FUNCTION_BLOCK FB_Sample EXTENDS FB_Generic
VAR_INPUT
END_VAR
VAR_OUTPUT
END_VAR
VAR
	lamp			: BOOL;	
	eStates			: E_SampleStates := E_SampleStates.IDLE;;
	eStateTemp		: E_SampleStates := E_SampleStates.IDLE;
	iStateTemp		: INT;	
END_VAR

SUPER^();
IF NOT subscribed THEN
	GVL.PubSubService.Subscribe(E_Topics.SAMPLE_SUBSCRRIBE_1,THIS^);
	GVL.PubSubService.Subscribe(E_Topics.SAMPLE_SUBSCRRIBE_2,THIS^);
	GVL.PubSubService.Subscribe(E_Topics.SAMPLE_SUBSCRRIBE_3,THIS^);
END_IF
subscribed	:= TRUE;


sComponent_name		:= 'fb_sample';
iComponetID			:= 99;
strState	:= ParseStateToString();

(*
Description: 
the callback that will be invoked when there is a publish for what the subscriber was subscribed to.
*)
METHOD Callback
VAR_INPUT
	data : PubSubData;
END_VAR
CASE data.Topic OF
	E_Topics.SAMPLE_SUBSCRRIBE_1:
		ADSLOGSTR(msgCtrlMask:= ADSLOG_MSGTYPE_LOG,msgFmtStr:='get data from publish 1',strArg:='');
	E_Topics.SAMPLE_SUBSCRRIBE_2:
		ADSLOGSTR(msgCtrlMask:= ADSLOG_MSGTYPE_LOG,msgFmtStr:='get data from publish 2',strArg:='');
	E_Topics.SAMPLE_SUBSCRRIBE_3:
		ADSLOGSTR(msgCtrlMask:= ADSLOG_MSGTYPE_LOG,msgFmtStr:='get data from publish 3',strArg:='');		
END_CASE
END_METHOD

{attribute 'object_name' := 'M_Aborting'}
METHOD M_Aborting
CASE fbUnitModeManager.eModeStatus OF	
	ePMLProtUnitMode_Production, ePMLProtUnitMode_Manual:		
		lamp	:= FALSE;		
		M_StateComplete();
			
	ePMLProtUnitMode_Maintenance, ePMLUnitMode_Service:
		
		M_StateComplete();
END_CASE
END_METHOD

METHOD M_agingTest : BOOL
VAR_INPUT
	
END_VAR
END_METHOD

{attribute 'object_name' := 'M_Completing'}
METHOD M_Completing
CASE fbUnitModeManager.eModeStatus OF
	ePMLProtUnitMode_Production:
		;
END_CASE
END_METHOD

{attribute 'object_name' := 'M_Execute'}
METHOD M_Execute

CASE fbUnitModeManager.eModeStatus OF
	ePMLProtUnitMode_Production:		//Mode Production
		//////////////////////////////////////////////////////////timeout//////////////////////////////////////////	
		iStateTemp	:= eStateTemp;
		ton_timeout();
		IF eStateTemp=eStates THEN
			ton_timeout.IN	:=TRUE;
		ELSE
			ton_timeout.IN	:=FALSE;
			eStateTemp	:= eStates;	
//			ParseStateToString();
//			GenerateErrorMsg(errorType:='M',strState:=ParseStateToString(),moduleID:=100,iState	:= iStateTemp);
			IF ton_timeout.Q THEN
				RETURN;
			END_IF
		END_IF
		IF ton_timeout.Q THEN	
			ton_timeout.IN	:=FALSE;
			CASE eStates OF	
				E_SampleStates.ERROR:	
					alarm_temp.Message	:= GenerateErrorMsg(errorType:='M',strState:=strState,iState := iStateTemp,errorMsg:='in error state.');
				ELSE
				alarm_temp.Message	:= GenerateErrorMsg(errorType:='M',strState:=strState,iState := iStateTemp,errorMsg:='time out');
			END_CASE
			
//			CASE eStates OF		
//				E_SampleStates.IDLE:						
//					;
//				E_SampleStates.INIT:
//					;
//				E_SampleStates.WAIT_ON:
//					;
//				E_SampleStates.WAIT_OFF:
//					;			
//				E_SampleStates.ERROR:	
//					alarm_temp.Message	:= 'Sample in error state';
//				ELSE
//					alarm_temp.Message	:= 'UNKNOWN STATES in Sample module';
//			END_CASE
			IF eStates<>E_SampleStates.IDLE AND eStates<>E_SampleStates.WAIT_ON AND eStates<>E_SampleStates.WAIT_OFF THEN
				GVL.pml_adminAlarm.M_SetAlarm(stAdmin:=GVL.PackTags.Admin,stAlarm:=alarm_temp);
			END_IF
		END_IF
		
		CASE eStates OF 
				E_SampleStates.IDLE:
					ton_timeout.PT	:= T#1MS;						
					eStates	:= E_SampleStates.INIT;				
				E_SampleStates.INIT:
					ton_timeout.PT	:= T#1S;
					eStates	:= E_SampleStates.WAIT_ON; 
				E_SampleStates.DETECTION:
					ton_timeout.PT	:= T#3S;
				E_SampleStates.WAIT:
					ton_timeout.PT	:= T#200MS;					
				E_SampleStates.WAIT_ON:
					lamp	:= TRUE;
					IF ton_timeout.Q THEN
						eStates	:= E_SampleStates.WAIT_OFF;
					END_IF
				E_SampleStates.WAIT_OFF:
					lamp	:= FALSE;
					IF ton_timeout.Q THEN
						eStates	:= E_SampleStates.IDLE;
					END_IF
				E_SampleStates.ERROR:
					;
			END_CASE
		
		
	ePMLProtUnitMode_Maintenance, ePMLUnitMode_Service:		
		//
		
	ePMLProtUnitMode_Manual:		//Manaul

END_CASE
END_METHOD

{attribute 'object_name' := 'M_Holding'}
METHOD M_Holding
CASE fbUnitModeManager.eModeStatus OF
	ePMLProtUnitMode_Production:		//Mode Production
		//Finisch the actual seperationstep	
		

	ePMLProtUnitMode_Maintenance:
		M_StateComplete();
END_CASE
END_METHOD

{attribute 'object_name' := 'M_Idle'}
METHOD M_Idle
IF G_HMI.bAging_test THEN
	//M_agingTest();
END_IF
END_METHOD

METHOD M_mapping : BOOL
VAR_INPUT
END_VAR
END_METHOD

METHOD M_Reset
VAR_INPUT
END_VAR
//Take away all commands
IF GVL.stChangeIntoProduction.bYesReset THEN
;
END_IF
END_METHOD

{attribute 'object_name' := 'M_Resetting'}
METHOD M_Resetting
CASE fbUnitModeManager.eModeStatus OF
	ePMLProtUnitMode_Production:		//Production, Mantainance, Manual
		lamp	:= FALSE;
		eStates :=E_SampleStates.IDLE;
		M_StateComplete();
	
	ePMLProtUnitMode_Maintenance, ePMLProtUnitMode_Manual, ePMLUnitMode_Service:
		M_StateComplete();
END_CASE
END_METHOD

{attribute 'object_name' := 'M_Starting'}
METHOD M_Starting
CASE fbUnitModeManager.eModeStatus OF
	ePMLProtUnitMode_Production:		//Production, Mantainance, Manual
		
		M_StateComplete();
	ePMLProtUnitMode_Maintenance, ePMLProtUnitMode_Manual, ePMLUnitMode_Service:
		M_StateComplete();
END_CASE
END_METHOD

{attribute 'object_name' := 'M_Stopping'}
METHOD M_Stopping
CASE fbUnitModeManager.eModeStatus OF
	ePMLProtUnitMode_Production, ePMLProtUnitMode_Manual:
				//////////////////////////////////////////////////////////timeout//////////////////////////////////////////	
		iStateTemp	:= eStateTemp;
		ton_timeout();
		IF eStateTemp=eStates THEN
			ton_timeout.IN	:=TRUE;
		ELSE
			ton_timeout.IN	:=FALSE;
			eStateTemp	:= eStates;	
		END_IF
		IF ton_timeout.Q THEN	
			ton_timeout.IN	:=FALSE;
			CASE eStates OF		
				E_SampleStates.IDLE:						
					;
				E_SampleStates.INIT:
					;
				E_SampleStates.WAIT_ON:
					;
				E_SampleStates.WAIT_OFF:
					;			
				E_SampleStates.ERROR:	
					alarm_temp.Message	:= 'Sample in error state';
				ELSE
					alarm_temp.Message	:= 'UNKNOWN STATES in Sample module';
			END_CASE
			IF eStates<>E_SampleStates.IDLE AND eStates<>E_SampleStates.WAIT_ON AND eStates<>E_SampleStates.WAIT_OFF THEN
				GVL.pml_adminAlarm.M_SetAlarm(stAdmin:=GVL.PackTags.Admin,stAlarm:=alarm_temp);
			END_IF
		END_IF
		
		CASE eStates OF 
				E_SampleStates.IDLE:						
					eStates	:= E_SampleStates.INIT;				
				E_SampleStates.INIT:
					ton_timeout.PT	:= T#1S;
					eStates	:= E_SampleStates.WAIT_ON; 
				E_SampleStates.WAIT_ON:
					lamp	:= TRUE;
					IF ton_timeout.Q THEN
						eStates	:= E_SampleStates.WAIT_OFF;
					END_IF
				E_SampleStates.WAIT_OFF:
					lamp	:= FALSE;
					IF ton_timeout.Q THEN
						eStates	:= E_SampleStates.IDLE;
						M_StateComplete();	
					END_IF
				E_SampleStates.ERROR:
					;
			END_CASE			
	ePMLProtUnitMode_Maintenance, ePMLUnitMode_Service:
		M_StateComplete();	
			//not defined
END_CASE
END_METHOD

{attribute 'object_name' := 'M_Undefined'}
METHOD M_Undefined

bUndefinedDone					:= TRUE;
END_METHOD

METHOD ParseStateToString : STRING
VAR_INPUT
END_VAR
CASE THIS^.eStates OF
	E_SampleStates.IDLE:
		ParseStateToString	:='IDLE';
	E_SampleStates.INIT:
		ParseStateToString	:='INIT';
	E_SampleStates.CHECK:
		ParseStateToString	:='CHECK';
	E_SampleStates.DETECTION:	
		ParseStateToString	:='DETECTION';
	E_SampleStates.LAMP_ON:
		ParseStateToString	:='LAMP_ON';
	E_SampleStates.LAMP_OFF:
		ParseStateToString	:='LAMP_OFF';
	E_SampleStates.WAIT:
		ParseStateToString	:='WAIT';
	E_SampleStates.WAIT_ON:
		ParseStateToString	:='WAIT_ON';
	E_SampleStates.WAIT_OFF:
		ParseStateToString	:='WAIT_OFF';
	E_SampleStates.DONE:	
		ParseStateToString	:='DONE';
	E_SampleStates.ERROR:
		ParseStateToString	:='ERROR';
	ELSE
		ParseStateToString	:='UNKNOW STATE';
END_CASE
END_METHOD

END_FUNCTION_BLOCK

(* stored: Version 1.1.0.1, ProductVersion 3.1.4024.12
   POU FB_Sample: Id {ac745d2e-72a6-4e96-8fa5-22b4fc8ce3be}, SpecialFunc None
   Method Callback: Id {13854ea2-63bf-4c04-b365-8df7edd8bd07}
   Method M_Aborting: Id {f930da81-89da-4559-a375-c186df3db1b8}
   Method M_agingTest: Id {9adad55d-8892-40fc-95e1-f07bfd3eee84}
   Method M_Completing: Id {1875369d-a175-4514-bc9e-11555728be77}
   Method M_Execute: Id {b3a6d44f-7c14-4bb5-8960-02311e08736a}
   Method M_Holding: Id {86cff955-61e4-408b-b2d8-f2046d06f0f0}
   Method M_Idle: Id {dfe9aba3-d5d0-42e7-b1ed-60e2c724fc75}
   Method M_mapping: Id {e0693328-8ff4-4bc0-a41b-371557aa2a9c}
   Method M_Reset: Id {f9a92c2c-cd0f-45e4-9799-65850bce3e92}
   Method M_Resetting: Id {4d657083-4b7f-4b47-b48f-38e10cf86d4a}
   Method M_Starting: Id {96856410-7941-4359-a2ce-673531411158}
   Method M_Stopping: Id {77c3cee3-a1f2-4fa1-aa43-d4090b723217}
   Method M_Undefined: Id {cdf2588c-c0af-48d6-a8bb-b7f419f8fb70}
   Method ParseStateToString: Id {5bca744c-9c54-4623-a6b9-77393438f207} *)
